FUNCTION_BLOCK Feeder (* Basic Function Block Type *)
  (* Standard: 61499-2 *)
  (* Version 0.0, 1/9/2024, Cheyan, Schneider Electric, Template *)
  PACKAGE Main;
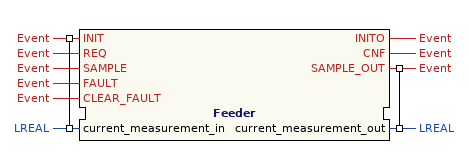
  EVENT_INPUT
    INIT WITH current_measurement_in;
    REQ;
    SAMPLE;
    FAULT;
    CLEAR_FAULT;
  END_EVENT
  EVENT_OUTPUT
    INITO; (* Initialization Confirm *)
    CNF; (* Execution Confirmation *)
    SAMPLE_OUT WITH current_measurement_out;
  END_EVENT
  VAR_INPUT
    current_measurement_in : LREAL; (* Input event qualifier *)
  END_VAR
  VAR_OUTPUT
    current_measurement_out : LREAL; (* Output event qualifier *)
  END_VAR
  VAR
    current_internal : LREAL;
  END_VAR
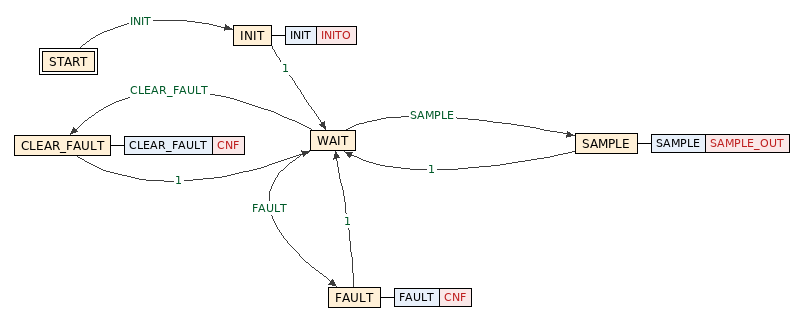
  EC_STATES
    START; (* Initial State *)
    INIT : INIT -> INITO; (* Initialization *)
    WAIT;
    SAMPLE : SAMPLE -> SAMPLE_OUT;
    FAULT : FAULT -> CNF;
    CLEAR_FAULT : CLEAR_FAULT -> CNF;
  END_STATES
  EC_TRANSITIONS
    INIT TO WAIT := 1;
    WAIT TO SAMPLE := SAMPLE;
    SAMPLE TO WAIT := 1;
    WAIT TO FAULT := FAULT;
    FAULT TO WAIT := 1;
    WAIT TO CLEAR_FAULT := CLEAR_FAULT;
    CLEAR_FAULT TO WAIT := 1;
    START TO INIT := INIT;
  END_TRANSITIONS
  ALGORITHM INIT IN ST: (* Initialization algorithm Setting the initial current measurement of the Feeder *)
;

current_internalnternal := current_measurement_in;
  END_ALGORITHM
  ALGORITHM REQ IN ST: (* Normally executed algorithm *)
;
  END_ALGORITHM
  ALGORITHM SAMPLE IN ST: (* Sending out current measurement *)
;

current_measurement_out := current_internal;
  END_ALGORITHM
  ALGORITHM FAULT IN ST: (* Triggering fault current. Fault current set at 1.5x of the normal current *)
;

current_internal := current_measurement_in + current_measurement_in/2;
  END_ALGORITHM
  ALGORITHM CLEAR_FAULT IN ST:
;

current_internal := 0;
  END_ALGORITHM
END_FUNCTION_BLOCK
